KUKA KRL program: hp235.src, hp235.dat

--- hp235.src ---
&ACCESS RVO
&COMMENT ANLAGE LEERFAHREN
&PARAM TEMPLATE = C:\KRC\ROBOTER\TEMPLATE\VG_HP
&PARAM EDITMASK = *
DEF hp235( )
;FOLD INI;%{PE}%V3.2.0,%MKUKATPBASIS,%CINIT,%VCOMMON,%P
;FOLD BAS INI;%{E}%V3.2.0,%MKUKATPBASIS,%CINIT,%VINIT,%P
GLOBAL INTERRUPT DECL 3 WHEN $STOPMESS==TRUE DO IR_STOPM ( )
INTERRUPT ON 3
BAS (#INITMOV,0 )
;ENDFOLD (BAS INI)
;FOLD GRIPPER INI;%{E}%V3.2.0,%MKUKATPGRIPPER,%CINIT,%VINIT,%P
USER_GRP(0,DUMMY,DUMMY,GDEFAULT)
;ENDFOLD (GRIPPER INI)
;FOLD SPOT INI;%{E}%V3.2.0,%MKUKATPSPOT,%CINIT,%VINIT,%P
USERSPOT(#INIT)
;ENDFOLD (SPOT INI)
;FOLD USER INI;%{E}%V3.2.0,%MKUKATPUSER,%CINIT,%VINIT,%P
;Make your modifications here
;FOLD COLLISION_V_3.00 INI ;%{E}
IF (COLLISION_DATA[1].I_NR>0) THEN
GLOBAL INTERRUPT DECL 21 WHEN $IN[COLLISION_DATA[1].I_NR]==FALSE DO COLLSTOP (1,0 )
ENDIF
IF (COLLISION_DATA[2].I_NR>0) THEN
GLOBAL INTERRUPT DECL 22 WHEN $IN[COLLISION_DATA[2].I_NR]==FALSE DO COLLSTOP (2,0 )
ENDIF
IF (COLLISION_DATA[3].I_NR>0) THEN
GLOBAL INTERRUPT DECL 23 WHEN $IN[COLLISION_DATA[3].I_NR]==FALSE DO COLLSTOP (3,0 )
ENDIF
IF (COLLISION_DATA[4].I_NR>0) THEN
GLOBAL INTERRUPT DECL 24 WHEN $IN[COLLISION_DATA[4].I_NR]==FALSE DO COLLSTOP (4,0 )
ENDIF
;ENDFOLD
;ENDFOLD (USER INI)
;ENDFOLD (INI)
;FOLD ; Anlagenbezeichn:               Stations-Nr:;%{PE}%R 3.2.24,%MKUKATPBASIS,%CCOMMENT,%VNORMAL,%P 2:Anlagenbezeichn:               Stations-Nr:
;ENDFOLD
;FOLD ; Stand / Version:;%{PE}%R 3.2.22,%MKUKATPBASIS,%CCOMMENT,%VNORMAL,%P 2:Stand / Version:
;ENDFOLD
;FOLD ; Name Bearbeiter:;%{PE}%R 3.2.22,%MKUKATPBASIS,%CCOMMENT,%VNORMAL,%P 2:Name Bearbeiter:
;ENDFOLD


;FOLD PTP HOME  Vel= 100 % DEFAULT;%{PE}%V3.2.0,%MKUKATPBASIS,%CMOVE,%VPTP,%P 1:PTP, 2:HOME, 3:, 5:100, 7:DEFAULT
$BWDSTART = FALSE
$H_POS=XHOME
PDAT_ACT=PDEFAULT
BAS (#PTP_DAT )
FDAT_ACT=FHOME
BAS (#FRAMES )
BAS (#VEL_PTP,100 )
PTP  XHOME
;ENDFOLD


;FOLD PTP HOME  Vel= 100 % DEFAULT;%{PE}%V3.2.0,%MKUKATPBASIS,%CMOVE,%VPTP,%P 1:PTP, 2:HOME, 3:, 5:100, 7:DEFAULT
$BWDSTART = FALSE
$H_POS=XHOME
PDAT_ACT=PDEFAULT
BAS (#PTP_DAT )
FDAT_ACT=FHOME
BAS (#FRAMES )
BAS (#VEL_PTP,100 )
PTP  XHOME
;ENDFOLD

END

--- hp235.dat ---
&ACCESS RVO
&COMMENT ANLAGE LEERFAHREN
&PARAM TEMPLATE = C:\KRC\ROBOTER\TEMPLATE\VG_HP
&PARAM EDITMASK = *
DEFDAT hp235
;FOLD EXTERNAL DECLARATIONS;%{PE}%V3.2.0,%MKUKATPBASIS,%CEXT,%VCOMMON,%P
;FOLD BAS EXT;%{PE}%V3.2.0,%MKUKATPBASIS,%CEXT,%VEXT,%P
EXT  BAS (BAS_COMMAND  :IN,REAL  :IN )
DECL INT SUCCESS
;ENDFOLD
;FOLD A10 EXT;%{E}%V3.2.0,%MKUKATPARC,%CEXT,%VEXT,%P
EXT  A10 (A_CMD_T:IN,A_STRT_T:IN,A_WELD_T:IN,A_END_T:IN,INT:IN)
;ENDFOLD
;FOLD A20 EXT;%{E}%V3.2.0,%MKUKATPA20,%CEXT,%VEXT,%P
EXT  A20 (INT  :IN,WELD_ST:IN,WELD_FI:IN,INT:IN)
;ENDFOLD
;FOLD GRIPPER EXT;%{E}%V3.2.0,%MKUKATPGRIPPER,%CEXT,%VEXT,%P
EXT  H50 (INT:IN, INT:IN ,INT:IN ,GRP_TYP:IN)
;ENDFOLD
;FOLD SPOT EXT;%{E}%V3.2.0,%MKUKATPSPOT,%CEXT,%VEXT,%P
EXT  USERSPOT (S_COMMAND  :IN, SPOT_TYPE:IN)
;ENDFOLD
;FOLD TOUCHSENSE EXT;%{E}%V3.2.0,%MKUKATPTS,%CEXT,%VEXT,%P
EXT  H70 (INT  :IN,SRCH_TYP_2  :OUT,E6POS  :IN,SRCH_TYP_3  :IN,SRCH_TYP_2  :IN,SRCH_TYP_2  :IN,SRCH_TYP_2  :IN,SRCH_TYP_2  :IN,SRCH_TYP_2  :IN,INT  :IN )
;ENDFOLD
;FOLD USER EXT;%{E}%V3.2.0,%MKUKATPUSER,%CEXT,%VEXT,%P
;Make here your modifications
;FOLD DC_BOLZEN_V3.00 ;%{}%V3.2.0,%MKUKATPUSER,%CEXT,%VEXT,%P
;EXT  BOLZEN (CALLMODE_T  :IN,INT  :IN,INT  :IN,INT  :IN,INT  :IN )
;ENDFOLD
;FOLD COLLISION_V3.00 ;%{}%V3.2.0,%MKUKATPUSER,%CEXT,%VEXT,%P
EXT  COLLSTOP (INT  :IN,INT  :IN )
;ENDFOLD
;ENDFOLD
;ENDFOLD

ENDDAT
